FUNCTION Fun_NumeroPiezasLadoCaballete : bool
VAR_INPUT
	NuPieasTotales 	: UINT ;
	PiezasLadoA		: POINTER TO UINT ;
	PiezasLadoB		: POINTER TO UINT ;
END_VAR
VAR
END_VAR

IF (NuPieasTotales MOD 2 = 1) THEN 
	PiezasLadoA^ := ( NuPieasTotales / 2) + 1  ;
	PiezasLadoB^ := ( NuPieasTotales / 2)  ;
ELSE
	PiezasLadoA^ := ( NuPieasTotales / 2)   ;
	PiezasLadoB^ := ( NuPieasTotales / 2)  ;
END_IF

END_FUNCTION

(* stored: Version 1.1.0.1, ProductVersion 3.1.4024.11
   POU Fun_NumeroPiezasLadoCaballete: Id {eedae483-f413-4a9d-90af-af392c8b6df9}, SpecialFunc None *)
